(* IEC 61131-3 sources: Docker-Support-and-Documentation/Examples/Automated Driveway, 3 files *)

(* ---- ACT.st ---- *)
tempIn := REAL_TO_INT(temp_inside / 10.0);
tempOut := REAL_TO_INT(temp_outside / 10.0);

//Exception in case of snow/ice
IF hour1.ice = TRUE OR hour2.ice = TRUE THEN
	PLC_PRG.exception := TRUE;
ELSE
	PLC_PRG.exception := FALSE;
END_IF

//If ground is wet, but might freeze later.
IF exception = FALSE AND hour1.rain > 0 AND hour1.temp > 0 THEN
	IF hour2.temp < 0 OR hour3.temp < 0 THEN
		PLC_PRG.exception := TRUE;
	ELSE
		PLC_PRG.exception := FALSE;
	END_IF
END_IF

//Normal conditions
IF hour1.rain > 0 AND hour1.temp < 0 THEN
	PLC_PRG.run := TRUE;
ELSE IF hour2.rain > 0 AND hour2.temp < 0 THEN
	 PLC_PRG.run := TRUE;
	 ELSE IF hour3.rain > 0 AND (tempOut <= -10 OR hour3.temp < -8) THEN
		PLC_PRG.run := TRUE;
		ELSE
			PLC_PRG.run := FALSE;
		END_IF
	 END_IF
END_IF

(*
IF IoConfig_Globals_Mapping.Port = TRUE THEN
	//TURN HEATER/OVEN OFF
END_IF *)

//MODE OF OPERATION
//MODE 1
IF PLC_PRG.mode1 = 1 THEN
	PLC_PRG.enable1 := 0;
	PLC_PRG.manual1 := FALSE;
	PLC_PRG.auto1 := FALSE;
ELSE IF PLC_PRG.mode1 = 2 THEN
		PLC_PRG.enable1 := TRUE;
		PLC_PRG.manual1 := TRUE;
		PLC_PRG.auto1 := FALSE;
	ELSE IF PLC_PRG.mode1 = 3 THEN
			PLC_PRG.enable1 := TRUE;
			PLC_PRG.manual1 := FALSE;
			PLC_PRG.auto1 := TRUE;
		END_IF
	END_IF
END_IF
//MODE 2
IF PLC_PRG.mode2 = 1 THEN
	PLC_PRG.enable2 := 0;
	PLC_PRG.manual2 := FALSE;
	PLC_PRG.auto2 := FALSE;
ELSE IF PLC_PRG.mode2 = 2 THEN
		PLC_PRG.enable2 := TRUE;
		PLC_PRG.manual2 := TRUE;
		PLC_PRG.auto2 := FALSE;
	ELSE IF PLC_PRG.mode2 = 3 THEN
			PLC_PRG.enable2 := TRUE;
			PLC_PRG.manual2 := FALSE;
			PLC_PRG.auto2 := TRUE;
		END_IF
	END_IF
END_IF
//MODE 3
IF PLC_PRG.mode3 = 1 THEN
	PLC_PRG.enable3 := 0;
	PLC_PRG.manual3 := FALSE;
	PLC_PRG.auto3 := FALSE;
ELSE IF PLC_PRG.mode3 = 2 THEN
		PLC_PRG.enable3 := TRUE;
		PLC_PRG.manual3 := TRUE;
		PLC_PRG.auto3 := FALSE;
	ELSE IF PLC_PRG.mode3 = 3 THEN
			PLC_PRG.enable3 := TRUE;
			PLC_PRG.manual3 := FALSE;
			PLC_PRG.auto3 := TRUE;
		END_IF
	END_IF
END_IF
//MODE 4
IF PLC_PRG.mode4 = 1 THEN
	PLC_PRG.enable4 := 0;
	PLC_PRG.manual4 := FALSE;
	PLC_PRG.auto4 := FALSE;
ELSE IF PLC_PRG.mode4 = 2 THEN
		PLC_PRG.enable4 := TRUE;
		PLC_PRG.manual4 := TRUE;
		PLC_PRG.auto4 := FALSE;
	ELSE IF PLC_PRG.mode4 = 3 THEN
			PLC_PRG.enable4 := TRUE;
			PLC_PRG.manual4 := FALSE;
			PLC_PRG.auto4 := TRUE;
		END_IF
	END_IF
END_IF

//Enabling auto
(*
IF PLC_PRG.auto1 = TRUE OR PLC_PRG.auto2 = TRUE OR PLC_PRG.auto3 = TRUE OR PLC_PRG.auto4 = TRUE THEN
	PLC_PRG.xEnableAuto := TRUE;
ELSE
	PLC_PRG.xEnableAuto := FALSE;
END_IF*)

//Power measurement
PLC_PRG.kWh1 := DWORD_TO_REAL(PLC_PRG.timeMin1)*300/(1000*60.0);
PLC_PRG.kWh2 := DWORD_TO_REAL(PLC_PRG.timeMin2)*300/(1000*60.0);
PLC_PRG.kWh3 := DWORD_TO_REAL(PLC_PRG.timeMin3)*300/(1000*60.0);
PLC_PRG.kWh4 := DWORD_TO_REAL(PLC_PRG.timeMin4)*300/(1000*60.0);
PLC_PRG.kWhTotal := PLC_PRG.kWh1 + PLC_PRG.kWh2 + PLC_PRG.kWh3 + PLC_PRG.kWh4 + kWh_charger;

(* ---- declarations.st ---- *)
PROGRAM PLC_PRG
VAR
	incomingRain : REAL;
	tempIn : INT;
	tempOut : INT;
	forecastTemp : INT;
	forecastRain : REAL;
	temp_inside	: REAL;
	temp_outside : REAL;

	xEnableManual : BOOL := FALSE;
	xEnableAuto : BOOL := FALSE;
	autoOn : BOOL;
	heatOn : BOOL;
	exception : BOOL;

	preTime : TIME := T#4H;   		//Predefined time for manual heating
	autoTime : TIME := T#90M; 		//Predefined time for when heating will start before snow/ice
	onTime : TIME;
	offTime : TIME;

	hour1 : WeatherData;
	hour2 : WeatherData;
	hour3 : WeatherData;
	hour4 : WeatherData;

	run : BOOL;
	manual1 : BOOL := FALSE;
	manual2 : BOOL := FALSE;
	manual3 : BOOL := FALSE;
	manual4 : BOOL := FALSE;
	enable1 : BOOL := TRUE;
	enable2 : BOOL := TRUE;
	enable3 : BOOL := TRUE;
	enable4 : BOOL := TRUE;
	auto1 : BOOL := TRUE;
	auto2 : BOOL := TRUE;
	auto3 : BOOL := TRUE;
	auto4 : BOOL := TRUE;
	mode1 : SINT := 3;
	mode2 : SINT := 3;
	mode3 : SINT := 3;
	mode4 : SINT := 3;
	(*
	DO1,DO2,DO3,DO4 : BOOL;
	DI1,DI2,DI3,DI4 : BOOL; *)

	auto: TOF;
	manTON: TON;
	manTON1: TON;
	manTON2: TON;
	manTON3: TON;
	manTON4: TON;
	F_TRIG_1: F_TRIG;
	F_TRIG_2: F_TRIG;
	F_TRIG_3: F_TRIG;
	F_TRIG_4: F_TRIG;
	F_TRIG_5: F_TRIG;
	timer1: WagoAppBuildingHVAC.FbOperatingHours_01;
	timer2: WagoAppBuildingHVAC.FbOperatingHours_01;
	timer3: WagoAppBuildingHVAC.FbOperatingHours_01;
	timer4: WagoAppBuildingHVAC.FbOperatingHours_01;
	charger_timer: WagoAppBuildingHVAC.FbOperatingHours_01;
	charger_powerMeasure: WagoAppPowerMeasurement.FbAC_Values_494;
	charger_powerTime: WagoAppBuildingHVAC.FbOperatingHours_01;

	powerMeter: BASIC.METER;
	reset_charger: BOOL;

	kW_Total : REAL;
	kW_Heating : REAL;
	kW_Charger : REAL;

END_VAR
VAR RETAIN PERSISTENT
	time1 : DWORD;
	time2 : DWORD;
	time3 : DWORD;
	time4 : DWORD;
	timeMin1 : DWORD;
	timeMin2 : DWORD;
	timeMin3 : DWORD;
	timeMin4 : DWORD;
	timeMin_charger: DWORD;
	kWh1 : REAL;
	kWh2 : REAL;
	kWh3 : REAL;
	kWh4 : REAL;
	kWh_Heating : REAL;
	kWh_Charger: REAL;
	kWh_Total : REAL;
END_VAR

(* ---- PLC_PRG.variables.iecst ---- *)
PROGRAM PLC_PRG
VAR
	incomingRain : REAL;
	tempIn : INT;
	tempOut : INT;
	forecastTemp : INT;
	forecastRain : REAL;

	xEnableManual : BOOL := FALSE;
	xEnableAuto : BOOL := FALSE;
	autoOn : BOOL;
	heatOn : BOOL;
	exception : BOOL;

	preTime : TIME := T#4H;   		//Predefined time for manual heating
	autoTime : TIME := T#90M; 		//Predefined time for when heating will start before snow/ice
	onTime : TIME;
	offTime : TIME;

	hour1 : WeatherData;
	hour2 : WeatherData;
	hour3 : WeatherData;
	hour4 : WeatherData;

	run : BOOL;
	manual1 : BOOL := FALSE;
	manual2 : BOOL := FALSE;
	manual3 : BOOL := FALSE;
	manual4 : BOOL := FALSE;
	enable1 : BOOL := TRUE;
	enable2 : BOOL := TRUE;
	enable3 : BOOL := TRUE;
	enable4 : BOOL := TRUE;
	auto1 : BOOL := TRUE;
	auto2 : BOOL := TRUE;
	auto3 : BOOL := TRUE;
	auto4 : BOOL := TRUE;
	mode1 : SINT := 3;
	mode2 : SINT := 3;
	mode3 : SINT := 3;
	mode4 : SINT := 3;

	auto: TOF;
	manTON: TON;
	manTON1: TON;
	manTON2: TON;
	manTON3: TON;
	manTON4: TON;
	F_TRIG_1: F_TRIG;
	F_TRIG_2: F_TRIG;
	F_TRIG_3: F_TRIG;
	F_TRIG_4: F_TRIG;
	F_TRIG_5: F_TRIG;
	timer1: WagoAppBuildingHVAC.FbOperatingHours_01;
	timer2: WagoAppBuildingHVAC.FbOperatingHours_01;
	timer3: WagoAppBuildingHVAC.FbOperatingHours_01;
	timer4: WagoAppBuildingHVAC.FbOperatingHours_01;
	charger_timer: WagoAppBuildingHVAC.FbOperatingHours_01;
	charger_powerMeasure: WagoAppPowerMeasurement.FbAC_Values_494;
	charger_powerTime: WagoAppBuildingHVAC.FbOperatingHours_01;

	powerMeter: BASIC.METER;
	reset_charger: BOOL;

END_VAR
VAR RETAIN PERSISTENT
	time1 : DWORD;
	time2 : DWORD;
	time3 : DWORD;
	time4 : DWORD;
	timeMin1 : DWORD;
	timeMin2 : DWORD;
	timeMin3 : DWORD;
	timeMin4 : DWORD;
	timeMin_charger: DWORD;
	kWh1 : REAL;
	kWh2 : REAL;
	kWh3 : REAL;
	kWh4 : REAL;
	kWh_charger: REAL;
	kWhTotal : REAL;
END_VAR
